// TIA Portal project "2022.06.04_星三角启动" (V17)

(* hardware
DEVICE "S7-1200 station_1"  S7-1200 Station
   slot 0: "Rack_0"  S7-1200 Rack  Rack  V1.0
   slot 1: "PLC_1"  CPU 1212C DC/DC/DC  6ES7 212-1AE40-0XB0  V4.5
*)

// ===== PLC "PLC_1"  CPU 1212C DC/DC/DC =====

VAR_GLOBAL   // PLC tag table "默认变量表"
   "启动" AT %I0.0 : Bool;
   "停止" AT %I0.1 : Bool;
   "主电源" AT %Q0.0 : Bool;
   "星形接触器" AT %Q0.1 : Bool;
   "三角形接触器" AT %Q0.2 : Bool;
   "Tag_1" AT %I0.2 : Bool;
   "Tag_2" AT %M0.0 : Bool;
   "Tag_3" AT %M0.1 : Bool;
END_VAR

// folder: System blocks/Program resources

DATA_BLOCK "IEC_Timer_0_DB"   // DB1
{ S7_Optimized_Access := 'TRUE' }
AUTHOR : Simatic
FAMILY : IEC
NAME : IEC_TMR
VERSION : 1.0
// stored: InstanceOfName IEC_TIMER
"IEC_TIMER"
BEGIN
END_DATA_BLOCK

DATA_BLOCK "IEC_Timer_0_DB_1"   // DB2
{ S7_Optimized_Access := 'TRUE' }
AUTHOR : Simatic
FAMILY : IEC
NAME : IEC_TMR
VERSION : 1.0
// stored: InstanceOfName IEC_TIMER
"IEC_TIMER"
BEGIN
END_DATA_BLOCK

// folder: (top level)

ORGANIZATION_BLOCK "Main"   // OB1, LAD, ProgramCycle
TITLE = "Main Program Sweep (Cycle)"
{ S7_Optimized_Access := 'TRUE' }
VERSION : 0.1
   VAR_INPUT
      Initial_Call : Bool;   // Initial call of this OB
      Remanence : Bool;   // =True, if remanent data are available
   END_VAR
BEGIN

REGION Network 1
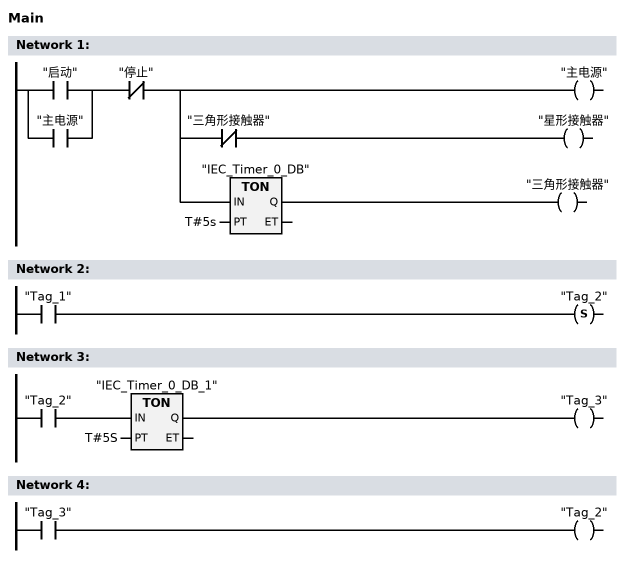
   "主电源" := ("启动" OR "主电源") AND NOT "停止";
   "星形接触器" := "主电源" AND NOT "三角形接触器";
   "IEC_Timer_0_DB".TON(IN := "主电源", PT := T#5s);
   "三角形接触器" := "IEC_Timer_0_DB".Q;
END_REGION

REGION Network 2
   RUNG wire#powerrail
      Contact( "Tag_1" )
      S_Coil( "Tag_2" )
   END_RUNG
   // the same network as SCL:
   IF "Tag_1" THEN "Tag_2" := TRUE; END_IF;
END_REGION

REGION Network 3
   "IEC_Timer_0_DB_1".TON(IN := "Tag_2", PT := T#5S);
   "Tag_3" := "IEC_Timer_0_DB_1".Q;
END_REGION

REGION Network 4
   RUNG wire#powerrail
      Contact( "Tag_3" )
      Coil( "Tag_2" )
   END_RUNG
   // the same network as SCL:
   "Tag_2" := "Tag_3";
END_REGION
END_ORGANIZATION_BLOCK